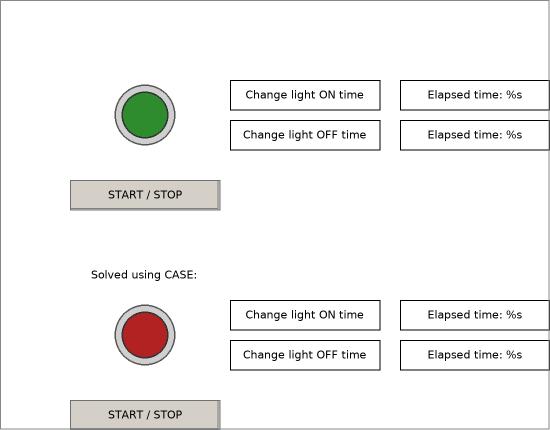
VISUALIZATION Visualization  // 550x430
    Lamp1 (110,80 70x70), variable: MAIN.fbBlinker.bLight, style: Lamp-Lamp1-Green
    Rectangle (230,80 150x30), "Change light ON time"
        OnMouseClick: write MAIN.dwTimeOn via Default
    Rectangle (230,120 150x30), "Change light OFF time"
        OnMouseClick: write MAIN.dwTimeOff via Default
    Button (70,180 150x30), "START / STOP"
        tap MAIN.bIsStartPressed
    Rectangle (400,80 150x30), "Elapsed time: %s", text variable: MAIN.fbBlinker.fbTimerOn.ET
    Rectangle (400,120 150x30), "Elapsed time: %s", text variable: MAIN.fbBlinker.fbTimerOff.ET
    Lamp1 (110,300 70x70), variable: MAIN.fbCaseBlinker.bLight, style: Lamp-Lamp1-Red
    Rectangle (230,300 150x30), "Change light ON time"
        OnMouseClick: write MAIN.dwCaseTimeOn via Default
    Rectangle (230,340 150x30), "Change light OFF time"
        OnMouseClick: write MAIN.dwCaseTimeOff via Default
    Button (70,400 150x30), "START / STOP"
        tap MAIN.bIsCaseStartPressed
    Rectangle (400,340 150x30), "Elapsed time: %s", text variable: MAIN.fbCaseBlinker.fbTimerOff.ET
    Rectangle (400,300 150x30), "Elapsed time: %s", text variable: MAIN.fbCaseBlinker.fbTimerOn.ET
    Rectangle (69,260 150x30), "Solved using CASE:"
END_VISUALIZATION

(* stored: Version 1.1.0.1, ProductVersion 3.1.4024.12
   Visu Visualization: Id {7b59bb49-7080-4193-87b7-35fdc16c5bcd} *)
